FUNCTION "Fx_Secret" : Void
{ S7_Optimized_Access := 'TRUE' }
VERSION : 0.1
   VAR_INPUT
      X : Int;
   END_VAR

   VAR_OUTPUT
      Y : Int;
   END_VAR


BEGIN
	// body is hidden by know-how protection in the fixture
	#Y := #X * 2;
END_FUNCTION
